// Mitsubishi GX Works2 project: pr6.1   PLC: Q03UDV

PROGRAM MAIN
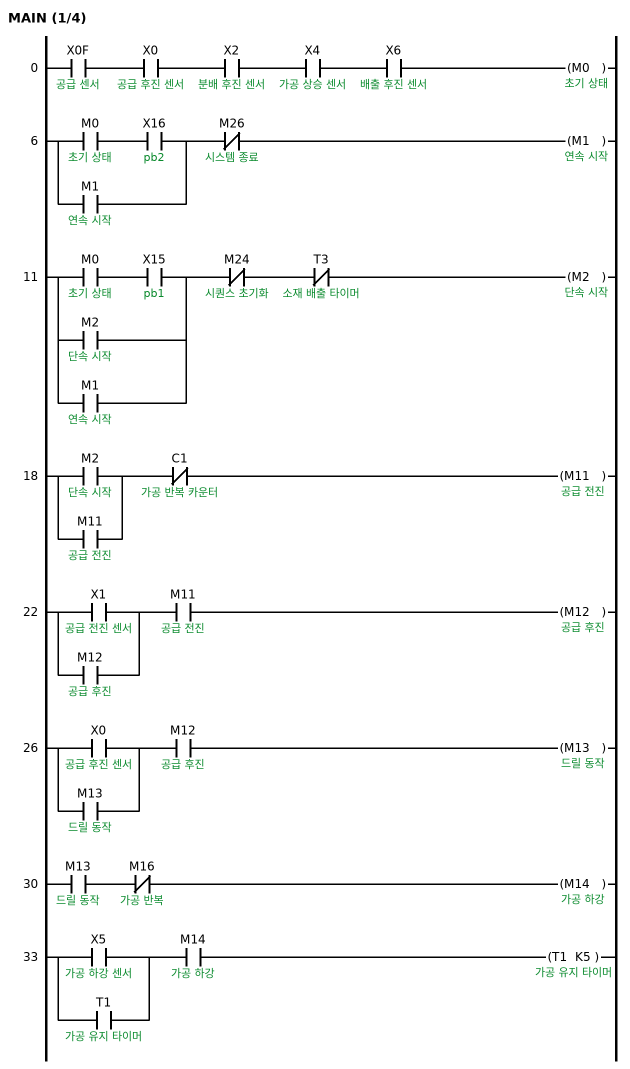
0     LD      X0F  ; 공급 센서
      AND     X0  ; 공급 후진 센서
      AND     X2  ; 분배 후진 센서
      AND     X4  ; 가공 상승 센서
      AND     X6  ; 배출 후진 센서
      OUT     M0  ; 초기 상태
6     LD      M0  ; 초기 상태
      AND     X16  ; pb2
      OR      M1  ; 연속 시작
      ANI     M26  ; 시스템 종료
      OUT     M1  ; 연속 시작
11    LD      M0  ; 초기 상태
      AND     X15  ; pb1
      OR      M2  ; 단속 시작
      OR      M1  ; 연속 시작
      ANI     M24  ; 시퀀스 초기화
      ANI     T3  ; 소재 배출 타이머
      OUT     M2  ; 단속 시작
18    LD      M2  ; 단속 시작
      OR      M11  ; 공급 전진
      ANI     C1  ; 가공 반복 카운터
      OUT     M11  ; 공급 전진
22    LD      X1  ; 공급 전진 센서
      OR      M12  ; 공급 후진
      AND     M11  ; 공급 전진
      OUT     M12  ; 공급 후진
26    LD      X0  ; 공급 후진 센서
      OR      M13  ; 드릴 동작
      AND     M12  ; 공급 후진
      OUT     M13  ; 드릴 동작
30    LD      M13  ; 드릴 동작
      ANI     M16  ; 가공 반복
      OUT     M14  ; 가공 하강
33    LD      X5  ; 가공 하강 센서
      OR      T1  ; 가공 유지 타이머
      AND     M14  ; 가공 하강
      OUT     T1 K5  ; 가공 유지 타이머
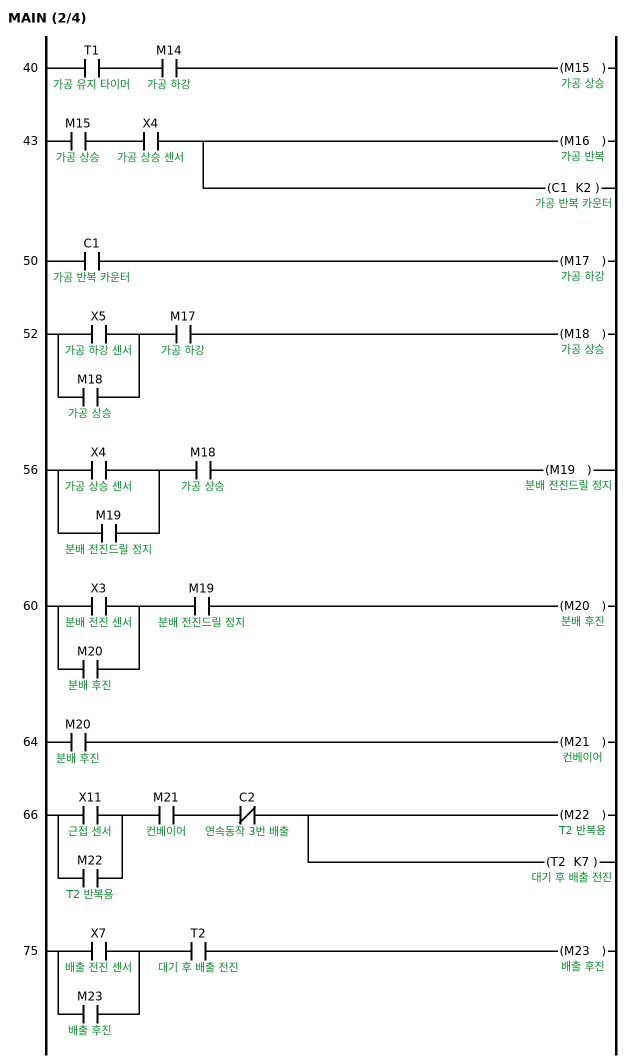
40    LD      T1  ; 가공 유지 타이머
      AND     M14  ; 가공 하강
      OUT     M15  ; 가공 상승
43    LD      M15  ; 가공 상승
      AND     X4  ; 가공 상승 센서
      OUT     M16  ; 가공 반복
      OUT     C1 K2  ; 가공 반복 카운터
50    LD      C1  ; 가공 반복 카운터
      OUT     M17  ; 가공 하강
52    LD      X5  ; 가공 하강 센서
      OR      M18  ; 가공 상승
      AND     M17  ; 가공 하강
      OUT     M18  ; 가공 상승
56    LD      X4  ; 가공 상승 센서
      OR      M19  ; 분배 전진드릴 정지
      AND     M18  ; 가공 상승
      OUT     M19  ; 분배 전진드릴 정지
60    LD      X3  ; 분배 전진 센서
      OR      M20  ; 분배 후진
      AND     M19  ; 분배 전진드릴 정지
      OUT     M20  ; 분배 후진
64    LD      M20  ; 분배 후진
      OUT     M21  ; 컨베이어
66    LD      X11  ; 근접 센서
      OR      M22  ; T2 반복용
      AND     M21  ; 컨베이어
      ANI     C2  ; 연속동작 3번 배출
      OUT     M22  ; T2 반복용
      OUT     T2 K7  ; 대기 후 배출 전진
75    LD      X7  ; 배출 전진 센서
      OR      M23  ; 배출 후진
      AND     T2  ; 대기 후 배출 전진
      OUT     M23  ; 배출 후진
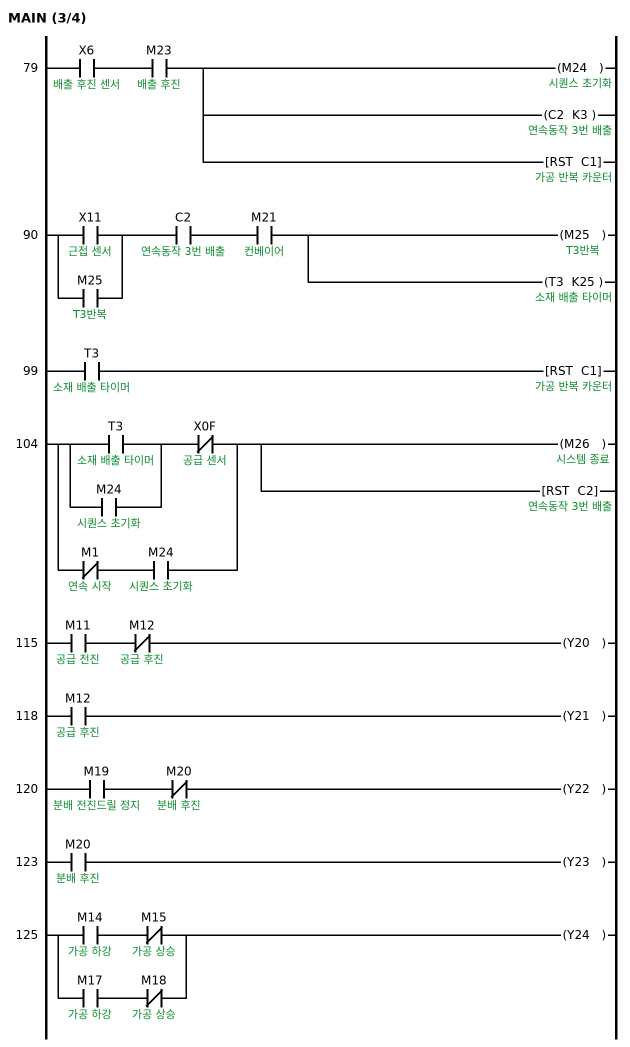
79    LD      X6  ; 배출 후진 센서
      AND     M23  ; 배출 후진
      OUT     M24  ; 시퀀스 초기화
      OUT     C2 K3  ; 연속동작 3번 배출
      RST     C1  ; 가공 반복 카운터
90    LD      X11  ; 근접 센서
      OR      M25  ; T3반복
      AND     C2  ; 연속동작 3번 배출
      AND     M21  ; 컨베이어
      OUT     M25  ; T3반복
      OUT     T3 K25  ; 소재 배출 타이머
99    LD      T3  ; 소재 배출 타이머
      RST     C1  ; 가공 반복 카운터
104   LD      T3  ; 소재 배출 타이머
      OR      M24  ; 시퀀스 초기화
      ANI     X0F  ; 공급 센서
      LDI     M1  ; 연속 시작
      AND     M24  ; 시퀀스 초기화
      ORB
      OUT     M26  ; 시스템 종료
      RST     C2  ; 연속동작 3번 배출
115   LD      M11  ; 공급 전진
      ANI     M12  ; 공급 후진
      OUT     Y20
118   LD      M12  ; 공급 후진
      OUT     Y21
120   LD      M19  ; 분배 전진드릴 정지
      ANI     M20  ; 분배 후진
      OUT     Y22
123   LD      M20  ; 분배 후진
      OUT     Y23
125   LD      M14  ; 가공 하강
      ANI     M15  ; 가공 상승
      LD      M17  ; 가공 하강
      ANI     M18  ; 가공 상승
      ORB
      OUT     Y24
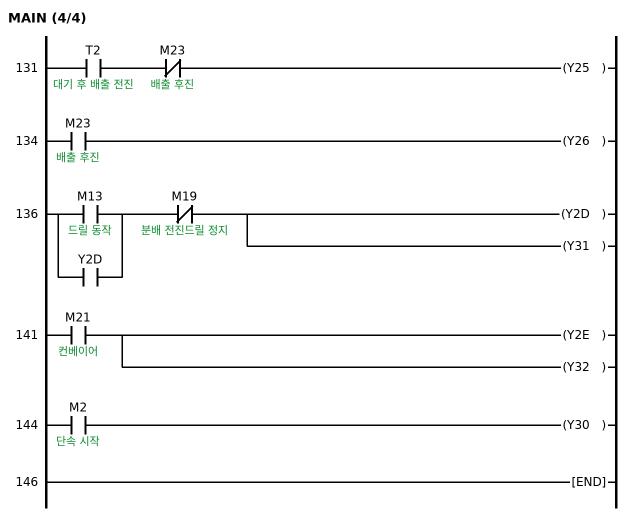
131   LD      T2  ; 대기 후 배출 전진
      ANI     M23  ; 배출 후진
      OUT     Y25
134   LD      M23  ; 배출 후진
      OUT     Y26
136   LD      M13  ; 드릴 동작
      OR      Y2D
      ANI     M19  ; 분배 전진드릴 정지
      OUT     Y2D
      OUT     Y31
141   LD      M21  ; 컨베이어
      OUT     Y2E
      OUT     Y32
144   LD      M2  ; 단속 시작
      OUT     Y30
146   END
END_PROGRAM

// device comments not shown above
M10  ; 작동 시작
M28  ; 드릴 정지
